Fanuc KAREL source: kb00065.KL

-- PROVISIONAL review KL for V1013-1; original PC SHA256 0524dcc69d95a81e4c044678810355b14dd9bc60d98db10372234c1dbf85837d
-- Incomplete behavior may be omitted. Consult companion uncertainty JSON. Do not deploy.
PROGRAM KB00065
%NOLOCKGROUP
BEGIN
  -- UNRESOLVED_PC offsets 5-14; opcodes 3F,75
  -- UNRESOLVED_PC offsets 19-26; opcodes 9D,23
  -- UNRESOLVED_PC offsets 31-38; opcodes 9D,23
  -- UNRESOLVED_PC offsets 43-52; opcodes 3F,75
  -- UNRESOLVED_PC offsets 57-66; opcodes 3F,75
  -- UNRESOLVED_PC offsets 71-78; opcodes 9D,23
  -- UNRESOLVED_PC offsets 83-90; opcodes 9D,23
  -- UNRESOLVED_PC offsets 95-102; opcodes 9D,23
  -- UNRESOLVED_PC offsets 107-165; opcodes 27,22,2A,22,22,22,2A,22,2A,22,22,22,31
  -- UNRESOLVED_PC offsets 170-174; opcodes 7F
END KB00065
